# EPICS IOC start-up script: test/startup/st.ymir-se-mc-mcu-01-epicscommodule.iocsh
require EthercatMC,USER

epicsEnvSet("MOTOR_PORT",    "$(SM_MOTOR_PORT=MCU1)")

epicsEnvSet("IPADDR",        "$(SM_IPADDR=172.30.244.59)")
epicsEnvSet("IPPORT",        "$(SM_IPPORT=5000)")
epicsEnvSet("ASYN_PORT",     "$(SM_ASYN_PORT=MC_CPU1)")
epicsEnvSet("PREFIX",        "$(SM_PREFIX=YMIR-SE:MC-MCU-01:)")
epicsEnvSet("PREC",          "$(SM_PREC=3)")
epicsEnvSet("SM_NOAXES",     "3")
epicsEnvSet("ECM_OPTIONS",   "adsPort=852"

< ethercatmcController.iocsh

#
# Axis 1
#
epicsEnvSet("AXISCONFIG",    "")
epicsEnvSet("MOTOR_NAME",    "m1")
epicsEnvSet("AXIS_NO",       "1")
epicsEnvSet("DESC",          "motor1")
< ethercatmcAxis.iocsh
< ethercatmcAxisdebug.iocsh
#< ethercatmcAxishome.iocsh

#
# Axis 2
#
epicsEnvSet("AXISCONFIG",    "")
epicsEnvSet("MOTOR_NAME",    "m2")
epicsEnvSet("AXIS_NO",       "2")
epicsEnvSet("DESC",          "motor2")
< ethercatmcAxis.iocsh
< ethercatmcAxisdebug.iocsh
#< ethercatmcAxishome.iocsh

#
# Axis 3
#
epicsEnvSet("AXISCONFIG",    "")
epicsEnvSet("MOTOR_NAME",    "m3")
epicsEnvSet("AXIS_NO",       "3")
epicsEnvSet("DESC",          "motor3")
< ethercatmcAxis.iocsh
< ethercatmcAxisdebug.iocsh
#< ethercatmcAxishome.iocsh
